// TIA Portal V20 export
TYPE "UDT_AnaMon08"
TITLE = MTPDataObjectSUCLibrary/DataAssembly/FlexAnaMon08
   STRUCT
      VSclMin { ExternalWritable := 'False'} : Real := 0.0;   // Value Scale Low Limit
      VSclMax { ExternalWritable := 'False'} : Real := 100.0;   // Value Scale High Limit
      VUnit { ExternalWritable := 'False'} : Int := 1001;   // Value Unit
      OSLevel : Byte := 16#00;   // OSLevel variable
      WQC { ExternalWritable := 'False'} : Byte := 16#FF;   // Worst Quality Code variable
      V { ExternalWritable := 'False'} : Real := 0.0;   // Value
      VLim1En { ExternalWritable := 'False'} : Bool;   // Enables Limit 11: enabled0: disabled
      VLim1 : Real;   // Limit 1 Value
      VLim1Act { ExternalWritable := 'False'} : Bool;   // Limit 1 active1: active0: inactive
      VMode1 { ExternalAccessible := 'False'; ExternalVisible := 'False'; ExternalWritable := 'False'} : Byte;   // Mode Limit 1
      VLim2En { ExternalWritable := 'False'} : Bool;   // Enables Limit 21: enabled0: disabled
      VLim2 : Real;   // Limit 2 Value
      VLim2Act { ExternalWritable := 'False'} : Bool;   // Limit 2 active1: active0: inactive
      VMode2 { ExternalAccessible := 'False'; ExternalVisible := 'False'; ExternalWritable := 'False'} : Byte;   // Mode Limit 2
      VLim3En { ExternalWritable := 'False'} : Bool;   // Enables Limit 31: enabled0: disabled
      VLim3 : Real;   // Limit 3 Value
      VLim3Act { ExternalWritable := 'False'} : Bool;   // Limit 3 active1: active0: inactive
      VMode3 { ExternalAccessible := 'False'; ExternalVisible := 'False'; ExternalWritable := 'False'} : Byte;   // Mode Limit 3
      VLim4En { ExternalWritable := 'False'} : Bool;   // Enables Limit 41: enabled0: disabled
      VLim4 : Real;   // Limit 4 Value
      VLim4Act { ExternalWritable := 'False'} : Bool;   // Limit 4 active1: active0: inactive
      VMode4 { ExternalAccessible := 'False'; ExternalVisible := 'False'; ExternalWritable := 'False'} : Byte;   // Mode Limit 4
      VLim5En { ExternalWritable := 'False'} : Bool;   // Enables Limit 51: enabled0: disabled
      VLim5 : Real;   // Limit 5 Value
      VLim5Act { ExternalWritable := 'False'} : Bool;   // Limit 5 active1: active0: inactive
      VMode5 { ExternalAccessible := 'False'; ExternalVisible := 'False'; ExternalWritable := 'False'} : Byte;   // Mode Limit 5
      VLim6En { ExternalWritable := 'False'} : Bool;   // Enables Limit 61: enabled0: disabled
      VLim6 : Real;   // Limit 6 Value
      VLim6Act { ExternalWritable := 'False'} : Bool;   // Limit 6 active1: active0: inactive
      VMode6 { ExternalAccessible := 'False'; ExternalVisible := 'False'; ExternalWritable := 'False'} : Byte;   // Mode Limit 6
      VLim7En { ExternalWritable := 'False'} : Bool;   // Enables Limit 71: enabled0: disabled
      VLim7 : Real;   // Limit 7 Value
      VLim7Act { ExternalWritable := 'False'} : Bool;   // Limit 7 active1: active0: inactive
      VMode7 { ExternalAccessible := 'False'; ExternalVisible := 'False'; ExternalWritable := 'False'} : Byte;   // Mode Limit 7
      VLim8En { ExternalWritable := 'False'} : Bool;   // Enables Limit 81: enabled0: disabled
      VLim8 : Real;   // Limit 8 Value
      VLim8Act { ExternalWritable := 'False'} : Bool;   // Limit 8 active1: active0: inactive
      VMode8 { ExternalAccessible := 'False'; ExternalVisible := 'False'; ExternalWritable := 'False'} : Byte;   // Mode Limit 8
   END_STRUCT;
END_TYPE
